TYPE U_TOUCH_PROBE_CTRL :
UNION
  stCtrl              : ARRAY[1..MAX_TOUCH_PROBE] OF ST_CTRL_TOUCH_PROBE;

  byCtrl    AT %I*    : ARRAY[1..MAX_TOUCH_PROBE] OF
                        ARRAY[1..SIZEOF(ST_CTRL_TOUCH_PROBE)] OF BYTE;
END_UNION
END_TYPE

(* stored: Version 1.1.0.1, ProductVersion 3.1.4026.13
   DUT U_TOUCH_PROBE_CTRL: Id {d3522c0b-542a-463f-b0d9-129aed8d68b0} *)
